(* IEC 61131-3 sources: POMIRTS_lab3/AS/Library_2/MTIdent/V1.10.0, 3 files *)

(* ---- MTIdent.typ ---- *)
(********************************************************************
 * COPYRIGHT -- Bernecker + Rainer
 ********************************************************************
 * Library: MTIdent
 * File: MTIdent.typ
 * Author: B&R
 * Created: August 30, 2013
 ********************************************************************
 * Data types of library MTIdent
 ********************************************************************)

TYPE
	MTIdentLSQInternalType : 	STRUCT
		CycleTime : REAL; (*Task cycle time. Unit: [s].*)
		ParametersValid : BOOL; (*Data for internal use.*)
		EnableOld : BOOL; (*Data for internal use.*)
		EnableDone : BOOL; (*Data for internal use.*)
		UpdateOld : BOOL; (*Data for internal use.*)
		DisabledBusy : BOOL; (*Data for internal use.*)
		StartIdentificationOld : BOOL; (*Data for internal use.*)
		SystemOrder : USINT; (*Order of numerator.*)
		WeightingFactor : REAL; (*Weighting factor.*)
		PMatrix : ARRAY[0..99]OF LREAL; (*Matrix for the recursive LSQ - algorithm.*)
		DataVector : ARRAY[0..9]OF LREAL; (*Data vector which contains the current input and output value of the plant as well as past values to compute the recursive LSQ algorithm.*)
		ParameterVector : ARRAY[0..9]OF LREAL; (*Estimated coefficients of the transfer function.*)
		NumberParameter : USINT; (*Number of parameter to be estimated.*)
		IdentificationState : USINT; (*Data for internal use.*)
		SettlingIndex : USINT; (*Data for internal use.*)
		NumberOfSettlingPhases : USINT; (*Data for internal use.*)
		LQParameterVector : ARRAY[0..2]OF REAL; (*Data for internal use.*)
		LQOutput : ARRAY[0..1]OF REAL; (*Data for internal use.*)
		StepHeight : REAL; (*Data for internal use.*)
		PlantOutputOld : REAL; (*Data for internal use.*)
		NoiseDeadBand : REAL; (*Data for internal use.*)
		PlantOutputOffset : REAL; (*Data for internal use.*)
		IdentificationSamples : USINT; (*Data for internal use.*)
		IdentificationDoneOld : BOOL; (*Data for internal use.*)
		SysRefParaNew : BOOL; (*Data for internal use.*)
		SampleTime : REAL; (*Data for internal use.*)
		CounterOld : UDINT; (*Data for internal use.*)
		SystemReference : MTTransferFcnType; (*Data for internal use.*)
	END_STRUCT;
END_TYPE

(* ---- MTIdent.fun ---- *)
(********************************************************************
 * COPYRIGHT -- Bernecker + Rainer
 ********************************************************************
 * Library: MTIdent
 * File: MTIdent.fun
 * Author: B&R
 * Created: August 30, 2013
 ********************************************************************
 * Functions and function blocks of library MTIdent
 ********************************************************************)

FUNCTION_BLOCK MTIdentLSQ (*This function block implements a recursive LSQ identification of a discrete dynamic system.*) (*$GROUP=User*)
	VAR_INPUT
		Enable : BOOL; (*Enable function block.*) (* *) (*#PAR#*)
		SystemOrder : USINT; (*System order of the parametric Model.*) (* *) (*#PAR#*)
		StepHeight : REAL; (*End value of the applied step for identification.*) (* *) (*#PAR#*)
		Update : BOOL; (*Parameters update trigger.*) (* *) (*#PAR#*)
		PlantOutput : REAL; (*Output signal of system.*) (* *) (*#CYC#*)
		StartIdentification : BOOL; (*Start and stop identification.*) (* *) (*#CMD#*)
		WeightingFactor : REAL; (*Weighting factor.*) (* *) (*#CMD#OPT#*)
	END_VAR
	VAR_OUTPUT
		Busy : BOOL; (*Function bolck is working.*) (* *) (*#PAR#*)
		Active : BOOL; (*Function block is active.*) (* *) (*#PAR#*)
		Error : BOOL; (*Indicates an error.*) (* *) (*#PAR#*)
		StatusID : DINT; (*Status information.*) (* *) (*#PAR#*)
		UpdateDone : BOOL; (*Update is sucessful.*) (* *) (*#PAR#*)
		PlantInput : REAL; (*Input signal for unkown system.*) (* *) (*#CYC#*)
		EstimationDeviation : REAL; (*Difference between the estimated and real plant output*) (* *) (*#CYC#*)
		IdentificationActive : BOOL; (*IdentificationActive denotes that the FB is identifying but can be stopped by the user any time.*) (* *) (*#CMD#*)
		IdentificationDone : BOOL; (*IdentificationDone recommends to use the identified data from up to now or even continue with the identification.*) (* *) (*#CMD#*)
		Numerator : ARRAY[0..4] OF REAL; (*Coefficients of numerator [b0, b1, b2, ... bm]. Maximum numerator order m = 4.*) (* *) (*#CMD#*)
		Denominator : ARRAY[0..5] OF REAL; (*Coefficients of denominator [a0, a1, a2, ... an]. Maximum denominator order n = 5.*) (* *) (*#CMD#*)
		SampleTime : REAL; (*SampleTime of transferfunction.*) (* *) (*#CMD#*)
		SystemReference : UDINT; (*System reference.*) (* *) (*#CMD#OPT#*)
	END_VAR
	VAR
		Internal : MTIdentLSQInternalType; (*Data for internal use.*)
	END_VAR
END_FUNCTION_BLOCK

(* ---- MTIdent.var ---- *)
(********************************************************************
 * COPYRIGHT -- Bernecker + Rainer
 ********************************************************************
 * Library: MTIdent
 * File: MTIdent.var
 * Author: B&R
 * Created: August 30, 2013
 ********************************************************************
 * Constants of library MTIdent
 ********************************************************************)
VAR CONSTANT
	mtACD_ERR_SYSTEM_ORDER_TOO_HIGH : DINT := -1058011144; (*Error: System order of parametric model invalid. Maximum SystemOrder= 5.*)
	mtACD_ERR_INVALID_SYSTEM_ORDER : DINT := -1058011143; (*Error: System order leads to a gain factor which is identified. Increas SystemOrder.*)
	mtACD_ERR_INVALID_WEIGHT_FACTOR : DINT := -1058011142; (*Error: WeightingFactor > 1 and < 0 not possible. Adjust WeightingFactor.*)
	mtACD_ERR_NOT_SETTLED_DOWN : DINT := -1058011141; (*Error: System is not settled down. Let oscillations fade away and try again.*)
	mtACD_WRN_SYSTEM_ORDER_TOO_HIGH : DINT := -2131752968; (*Warning: System order of parametric model invalid. Maximum SystemOrder= 5.*)
	mtACD_WRN_INVALID_SYSTEM_ORDER : DINT := -2131752967; (*Warning: System order leads to a gain factor which is identified. Increase SystemOrder.*)
	mtACD_WRN_INVALID_WEIGHT_FACTOR : DINT := -2131752966; (*Warning: WeightingFactor > 1 and < 0 not possible. Adjust WeightingFactor.*)
	mtACD_WRN_SMALL_WEIGHT_FACTOR : DINT := -2131752965; (*Warning: Small WeightingFactor may lead to bad results.*)
	mtACD_WRN_NOT_SETTLED_DOWN : DINT := -2131752964; (*Warning: System is not settled down. Let oscillations fade away and try again.*)
	mtACD_WRN_ABORTED_TOO_EARLY : DINT := -2131752963; (*Warning: Identification was aborted too early.*)
	mtACD_WRN_OTHER_FB_USES_SYSREF : DINT := -2131755008; (*Warning: Another function block is using the data for this system reference.*)
END_VAR
